// TIA Portal project "Ex2-PickAndPlace" (V16)
// The pick and place project

(* hardware
DEVICE "S7-1200 station_1"  S7-1200 Station
   slot 0: "Rack_0"  S7-1200 Rack  Rack  V1.0
   slot 1: "PLC_1"  CPU 1215C DC/DC/Rly  6ES7 215-1HG40-0XB0  V4.4
*)

// ===== PLC "PLC_1"  CPU 1215C DC/DC/Rly =====

VAR_GLOBAL   // PLC tag table "Default tag table"
   "System_Byte" AT %MB254 : Byte;
   "FirstScan" AT %M254.0 : Bool;
   "DiagStatusUpdate" AT %M254.1 : Bool;
   "AlwaysTRUE" AT %M254.2 : Bool;
   "AlwaysFALSE" AT %M254.3 : Bool;
   "Clock_Byte" AT %MB255 : Byte;
   "Clock_10Hz" AT %M255.0 : Bool;
   "Clock_5Hz" AT %M255.1 : Bool;
   "Clock_2.5Hz" AT %M255.2 : Bool;
   "Clock_2Hz" AT %M255.3 : Bool;
   "Clock_1.25Hz" AT %M255.4 : Bool;
   "Clock_1Hz" AT %M255.5 : Bool;
   "Clock_0.625Hz" AT %M255.6 : Bool;
   "Clock_0.5Hz" AT %M255.7 : Bool;
END_VAR

// folder: DB's

DATA_BLOCK "FB_CM_DI_Sensor_DB"   // DB1
{ S7_Optimized_Access := 'FALSE' }
AUTHOR : GeertVG
FAMILY : S88
VERSION : 0.1
// stored: InstanceOfName FB_CM_DI_Sensor
"FB_CM_DI_Sensor"
BEGIN
END_DATA_BLOCK

DATA_BLOCK "FB_PE_StartStop_DB"   // DB11
{ S7_Optimized_Access := 'FALSE' }
AUTHOR : GeertVG
FAMILY : S88
VERSION : 0.1
// stored: InstanceOfName FB_PE_StartStop
"FB_PE_StartStop"
BEGIN
END_DATA_BLOCK

DATA_BLOCK "FB_PE_Reset_DB"   // DB12
{ S7_Optimized_Access := 'FALSE' }
AUTHOR : GeertVG
FAMILY : S88
VERSION : 0.1
// stored: InstanceOfName FB_PE_Reset
"FB_PE_Reset"
BEGIN
END_DATA_BLOCK

DATA_BLOCK "FB_CM_Lamp_DB"   // DB13
{ S7_Optimized_Access := 'FALSE' }
AUTHOR : GeertVG
FAMILY : S88
VERSION : 0.1
// stored: InstanceOfName FB_CM_Lamp
"FB_CM_Lamp"
BEGIN
END_DATA_BLOCK

// folder: (top level)

FUNCTION_BLOCK "S88"   // FB1, FBD
TITLE = S88
{ S7_Optimized_Access := 'TRUE' }
VERSION : 0.1
// S88 software model for the pick and place project
BEGIN

REGION Network 1: Control module sensor
END_REGION
END_FUNCTION_BLOCK

FUNCTION "FC_EM_PnP" : Void   // FC1, FBD
TITLE = Equipment module for the pick and place
{ S7_Optimized_Access := 'TRUE' }
VERSION : 0.1
// Equipment module following the S88 software model for the pick and place project
BEGIN

REGION Network 1: Control module sensor B1
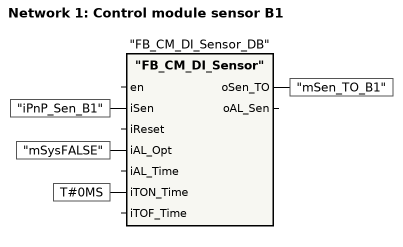
   "FB_CM_DI_Sensor_DB"(iSen := "iPnP_Sen_B1",   // "FB_CM_DI_Sensor"
                        iAL_Opt := "mSysFALSE",
                        iTON_Time := T#0MS,
                        oSen_TO => "mSen_TO_B1");
END_REGION
END_FUNCTION

FUNCTION "FC_EM_CC1" : Void   // FC2, FBD
TITLE = Circuit board 1
{ S7_Optimized_Access := 'TRUE' }
VERSION : 0.1
// This cicruit board handles the start and stop instruction. Lamps are being controlled here as well
BEGIN

REGION Network 1: Procedure element start stop
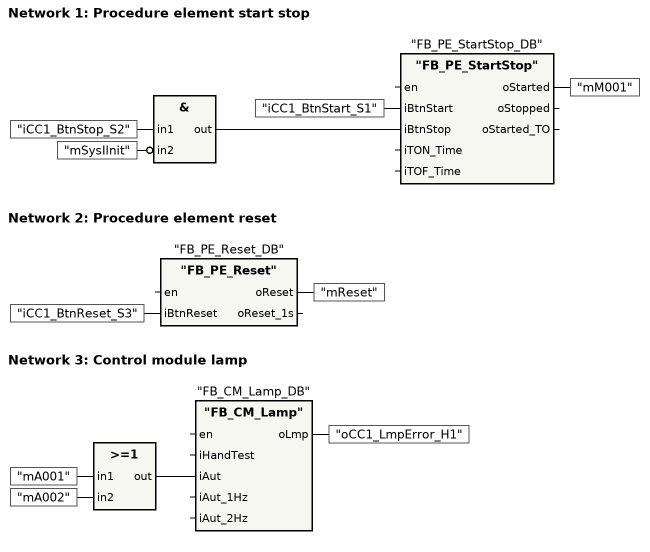
   "FB_PE_StartStop_DB"(iBtnStart := "iCC1_BtnStart_S1",   // "FB_PE_StartStop"
                        iBtnStop := "iCC1_BtnStop_S2" AND NOT "mSysIlnit",
                        oStarted => "mM001");
END_REGION

REGION Network 2: Procedure element reset
   "FB_PE_Reset_DB"(iBtnReset := "iCC1_BtnReset_S3", oReset => "mReset");   // "FB_PE_Reset"
END_REGION

REGION Network 3: Control module lamp
   "FB_CM_Lamp_DB"(iAut := "mA001" OR "mA002", oLmp => "oCC1_LmpError_H1");   // "FB_CM_Lamp"
END_REGION
END_FUNCTION

ORGANIZATION_BLOCK "Main"   // OB1, FBD, ProgramCycle
TITLE = "Main Program Sweep (Cycle)"
{ S7_Optimized_Access := 'TRUE' }
VERSION : 0.1
   VAR_INPUT
      Initial_Call : Bool;   // Initial call of this OB
      Remanence : Bool;   // =True, if remanent data are available
   END_VAR
BEGIN

REGION Network 1
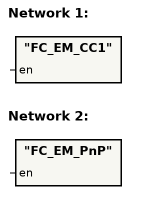
   "FC_EM_CC1"();
END_REGION

REGION Network 2
   "FC_EM_PnP"();
END_REGION
END_ORGANIZATION_BLOCK

// folder: Control modules (CM)

FUNCTION_BLOCK "FB_CM_DI_Sensor"   // FB10, FBD
TITLE = Control module digital sensor
{ S7_Optimized_Access := 'FALSE' }
AUTHOR : GeertVG
FAMILY : S88
VERSION : 0.1
// A control modul digital sensor processes the signal coming from a digital sensor and can delay a signal with the use of a rise- or a switch-off delay and/or in case a sensor gets activated to activate an alarm.
   VAR_INPUT
      iSen : Bool;   // Sensor
      iReset : Bool;   // Reset alarm
      iAL_Opt : Bool;   // Alarm option enabled if TRUE
      iAL_Time : Time;   // Rise-delay sensor alarm
      iTON_Time : Time;   // Sensor rise-delay
      iTOF_Time : Time;   // Sensor switch-off delay
   END_VAR
   VAR_OUTPUT
      oSen_TO : Bool;   // Sensor after delay
      oAL_Sen : Bool;   // Alarm sensor activated
   END_VAR
   VAR
      sTON_AL : TON_TIME;   // Rise-delay for oAL_sen
      sTON : TON_TIME;   // Rise-delay for oSen_TO
      sTOF : TOF_TIME;   // Switch-off delay for oSen_TO
      sAL_Sen : Bool;   // Sensor alarm
      sTON_Aon : Bool;
   END_VAR
BEGIN

REGION Network 1: Rise-delay for the activated alarm sensor
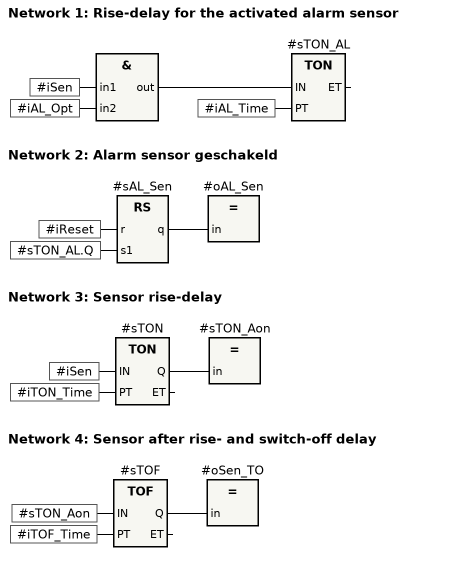
   #sTON_AL(IN := #iSen AND #iAL_Opt, PT := #iAL_Time);   // TON
END_REGION

REGION Network 2: Alarm sensor geschakeld
   IF #iReset THEN
       #sAL_Sen := FALSE;   // RS flip-flop
   END_IF;
   IF #sTON_AL.Q THEN #sAL_Sen := TRUE; END_IF;
   #oAL_Sen := #sAL_Sen;
END_REGION

REGION Network 3: Sensor rise-delay
   #sTON(IN := #iSen, PT := #iTON_Time);   // TON
   #sTON_Aon := #sTON.Q;
END_REGION

REGION Network 4: Sensor after rise- and switch-off delay
   #sTOF(IN := #sTON_Aon, PT := #iTOF_Time);   // TOF
   #oSen_TO := #sTOF.Q;
END_REGION
END_FUNCTION_BLOCK

FUNCTION_BLOCK "FB_CM_Lamp"   // FB16, FBD
TITLE = Control module lamp
{ S7_Optimized_Access := 'FALSE' }
AUTHOR : GeertVG
FAMILY : S88
VERSION : 0.1
// A control module lamp will actiavte a lamp (if chosen blinking). Also the possibility of testing the lamp with the use of the test input.
   VAR_INPUT
      iHandTest : Bool;   // Lamptest
      iAut : Bool;   // Lamp continue activation
      iAut_1Hz : Bool;   // Lamp blinking slowly
      iAut_2Hz : Bool;   // Lamp blinking fast
   END_VAR
   VAR_OUTPUT
      oLmp : Bool;   // Lamp
   END_VAR
   VAR
      sTON_1Hz_On : TON_TIME;   // 1 Hz timer lamp on
      sTON_1Hz_Off : TON_TIME;   // 1 Hz timer lamp off
      sTON_2Hz_On : TON_TIME;   // 2 Hz timer lamp on
      sTON_2Hz_Off : TON_TIME;   // 2 Hz timer lamp off
      sOn_1Hz : Bool;
      sOff_1Hz : Bool;
      sOn_2Hz : Bool;
      sOff_2Hz : Bool;
   END_VAR
BEGIN

REGION Network 1: Blinkcicuit 1Hz
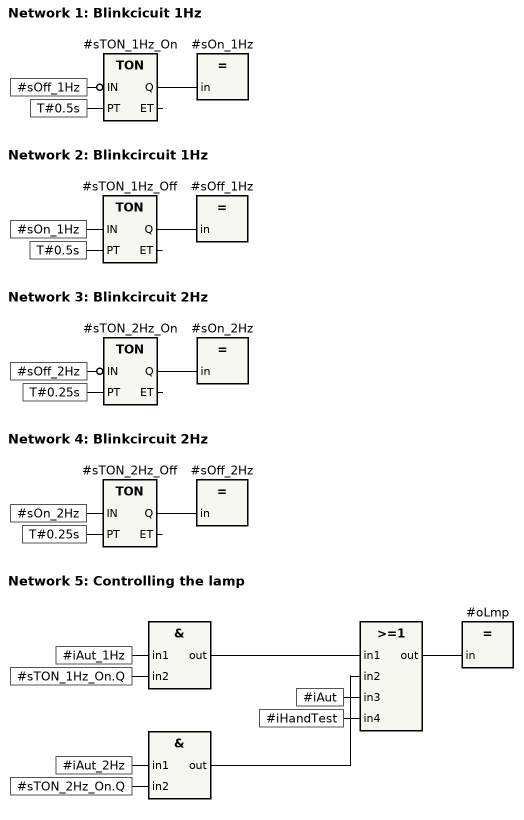
   #sTON_1Hz_On(IN := NOT #sOff_1Hz, PT := T#0.5s);   // TON
   #sOn_1Hz := #sTON_1Hz_On.Q;
END_REGION

REGION Network 2: Blinkcircuit 1Hz
   #sTON_1Hz_Off(IN := #sOn_1Hz, PT := T#0.5s);   // TON
   #sOff_1Hz := #sTON_1Hz_Off.Q;
END_REGION

REGION Network 3: Blinkcircuit 2Hz
   #sTON_2Hz_On(IN := NOT #sOff_2Hz, PT := T#0.25s);   // TON
   #sOn_2Hz := #sTON_2Hz_On.Q;
END_REGION

REGION Network 4: Blinkcircuit 2Hz
   #sTON_2Hz_Off(IN := #sOn_2Hz, PT := T#0.25s);   // TON
   #sOff_2Hz := #sTON_2Hz_Off.Q;
END_REGION

REGION Network 5: Controlling the lamp
   #oLmp := (#iAut_1Hz AND #sTON_1Hz_On.Q) OR (#iAut_2Hz AND #sTON_2Hz_On.Q) OR #iAut OR #iHandTest;
END_REGION
END_FUNCTION_BLOCK

// folder: Procedure Elements (PE)

FUNCTION_BLOCK "FB_PE_StartStop"   // FB30, FBD
TITLE = Start-Stop procedure element
{ S7_Optimized_Access := 'FALSE' }
AUTHOR : GeertVG
FAMILY : S88
VERSION : 0.1
// A start-stop is used to start and stop actuators and/or the automatic process of a installation/machine (or parts of it).
   VAR_INPUT
      iBtnStart : Bool;   // Start button(NO)
      iBtnStop : Bool;   // Stop button (NC)
      iTON_Time : Time;   // Opkomvertraging voor oGestart_TO
      iTOF_Time : Time;   // Afvalvertraging voor oGestart_TO
   END_VAR
   VAR_OUTPUT
      oStarted : Bool;   // Started
      oStopped : Bool;   // Stopped
      oStarted_TO : Bool;   // Started with a rise or off-delay
   END_VAR
   VAR
      sStarted : Bool;   // Started
      sPfBtnStart : Bool;   // Rising flank of iBtnStart
      sTON_Started : Bool;   // Start with on-delay
      sTON : TON_TIME;   // On-delay
      sTOF : TOF_TIME;   // Off-delay
   END_VAR
   VAR_TEMP   // added for the SCL form of the ladder/FBD networks
      _w1 : Bool;
   END_VAR
BEGIN

REGION Network 1: Start-stop using a FlipFlop instruction
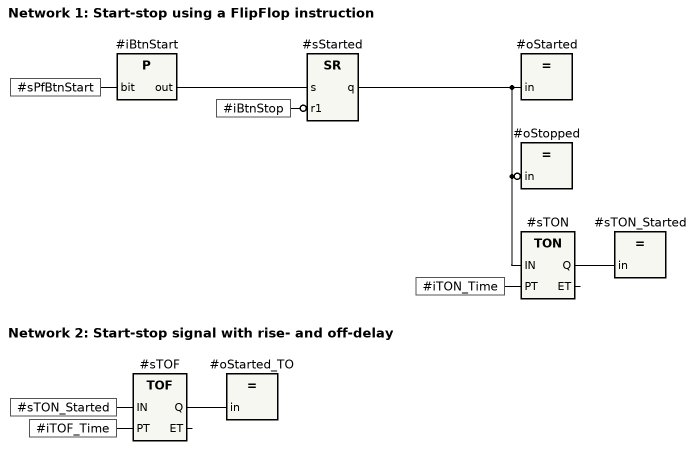
   #_w1 := #iBtnStart AND NOT #sPfBtnStart;   // rising edge of #iBtnStart
   #sPfBtnStart := #iBtnStart;
   IF #_w1 THEN
       #sStarted := TRUE;   // SR flip-flop
   END_IF;
   IF NOT #iBtnStop THEN #sStarted := FALSE; END_IF;
   #oStarted := #sStarted;
   #oStopped := NOT #sStarted;
   #sTON(IN := #sStarted, PT := #iTON_Time);   // TON
   #sTON_Started := #sTON.Q;
END_REGION

REGION Network 2: Start-stop signal with rise- and off-delay
   #sTOF(IN := #sTON_Started, PT := #iTOF_Time);   // TOF
   #oStarted_TO := #sTOF.Q;
END_REGION
END_FUNCTION_BLOCK

FUNCTION_BLOCK "FB_PE_Reset"   // FB31, FBD
TITLE = Reset procedure element
{ S7_Optimized_Access := 'FALSE' }
AUTHOR : GeertVG
FAMILY : S88
VERSION : 0.1
// The reset procedure is commonly used to create a controlled reset signal. Controlled because the signal is coming from a for example. an electyrical reset button (NO contact) can contain errors like a shortcircuit, the bridging of a signal and a bad/ fake contact.
   VAR_INPUT
      iBtnReset : Bool;   // Reset button
   END_VAR
   VAR_OUTPUT
      oReset : Bool;   // Checked reset signal (1 cyclus)
      oReset_1s : Bool;   // Checked reset signal (1s)
   END_VAR
   VAR
      sNfReset : Bool;
      sTON_Max : TON_TIME;   // Max. time that the button can be pressed
      sTON_Min : TON_TIME;   // Min. time that the button can be pressed
      sTP : TP_TIME;   // Checked reset time off 1s
   END_VAR
   VAR_TEMP   // added for the SCL form of the ladder/FBD networks
      _w1 : Bool;
   END_VAR
BEGIN

REGION Network 1: Max. time
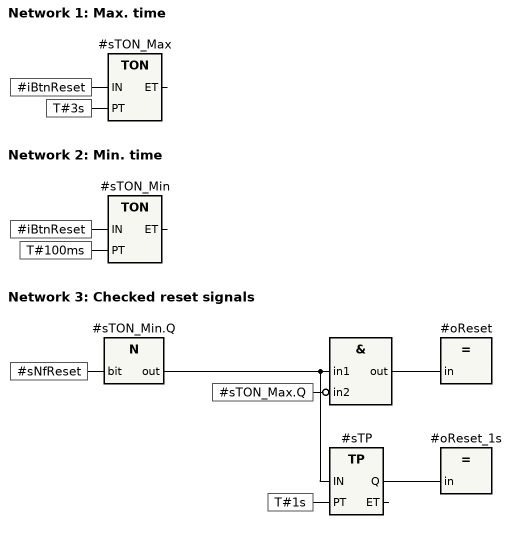
   #sTON_Max(IN := #iBtnReset, PT := T#3s);   // TON
END_REGION

REGION Network 2: Min. time
   #sTON_Min(IN := #iBtnReset, PT := T#100ms);   // TON
END_REGION

REGION Network 3: Checked reset signals
   #_w1 := NOT #sTON_Min.Q AND #sNfReset;   // falling edge of #sTON_Min.Q
   #sNfReset := #sTON_Min.Q;
   #oReset := #_w1 AND NOT #sTON_Max.Q;
   #sTP(IN := #_w1, PT := T#1s);   // TP
   #oReset_1s := #sTP.Q;
END_REGION
END_FUNCTION_BLOCK

// ===== library types =====

// folder: Control modules (CM)

FUNCTION_BLOCK "FB_CM_AI_Sensor"   // FB11, FBD
TITLE = Control module analogesensor
{ S7_Optimized_Access := 'FALSE' }
AUTHOR : GeertVG
FAMILY : S88
VERSION : 0.1
// The control module analog sensor converts a measured number to a SI-Unit
// In case of incorrect operation of the sensor a alarm will be created.
   VAR_INPUT
      iSen : Int;   // Measured value
      iReset : Bool;   // Reset alarm
      iHiLim : Real;   // The upper measurelimit of the sensor
      iLoLim : Real;   // The lower measurelimit of the sensor
      iUniOpt : Bool;   // 1 = Unipolair / 0 = Bipolair
   END_VAR
   VAR_OUTPUT
      oX : Real;   // The measured value gets converted to a SI-Unit
      oAL_Sen : Bool;   // Alarm sensor defect
   END_VAR
   VAR
      sAL_Sen : Bool;   // Alarm sensor defect
      sSen_DINT : DInt;   // Measured Value
      sMIN : DInt;   // Under Limit
      sNORM_Counter : DInt;
      sNORM_Denominator : DInt;
      sNORM_Counter_REAL : Real;
      sNORM_Denominator_REAL : Real;
      sNORM_X : Real;
      sSCALE_MeasureRange : Real;
      sSCALE_X : Real;
   END_VAR
BEGIN

REGION Network 1: Conversion sensor
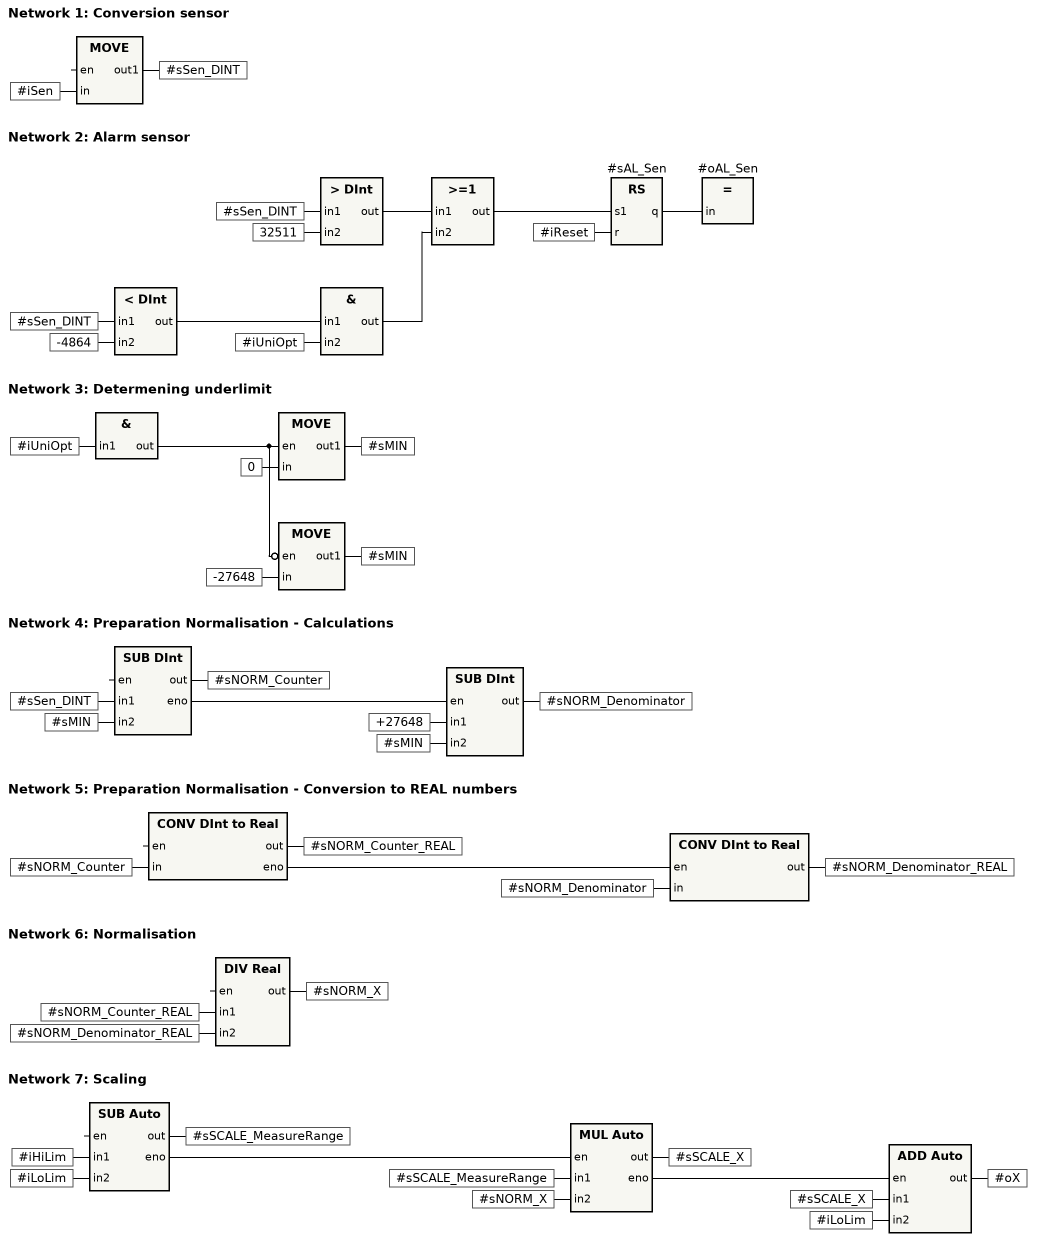
   #sSen_DINT := #iSen;
END_REGION

REGION Network 2: Alarm sensor
   IF #iReset THEN
       #sAL_Sen := FALSE;   // RS flip-flop
   END_IF;
   IF (#sSen_DINT > 32511) OR ((#sSen_DINT < (-4864)) AND #iUniOpt) THEN #sAL_Sen := TRUE; END_IF;
   #oAL_Sen := #sAL_Sen;
END_REGION

REGION Network 3: Determening underlimit
   IF #iUniOpt THEN #sMIN := 0; END_IF;
   IF NOT #iUniOpt THEN #sMIN := -27648; END_IF;
END_REGION

REGION Network 4: Preparation Normalisation - Calculations
   #sNORM_Counter := #sSen_DINT - #sMIN;
   #sNORM_Denominator := +27648 - #sMIN;
END_REGION

REGION Network 5: Preparation Normalisation - Conversion to REAL numbers
   #sNORM_Counter_REAL := DINT_TO_REAL(#sNORM_Counter);
   #sNORM_Denominator_REAL := DINT_TO_REAL(#sNORM_Denominator);
END_REGION

REGION Network 6: Normalisation
   #sNORM_X := #sNORM_Counter_REAL / #sNORM_Denominator_REAL;
END_REGION

REGION Network 7: Scaling
   #sSCALE_MeasureRange := #iHiLim - #iLoLim;
   #sSCALE_X := #sSCALE_MeasureRange * #sNORM_X;
   #oX := #sSCALE_X + #iLoLim;
END_REGION
END_FUNCTION_BLOCK

FUNCTION_BLOCK "FB_CM_DOL"   // FB12, FBD
TITLE = Control module asynchronous motor 1 direction 1 speed
{ S7_Optimized_Access := 'FALSE' }
AUTHOR : GeertVG
FAMILY : S88
VERSION : 0.1
// A control module asynchronous motor 1 direction 1 speed controls the management of a 3-phase asynchronous motor with a motor circuit breaker and one contactor. The control module is provided with a hand workmode, an automatic workingmode, moter circuit breaker alarm and an enable.
   VAR_INPUT
      iEnable : Bool;
      iReset : Bool;
      iMcb : Bool;
      iModeHand : Bool;
      iHandOn : Bool;
      iHandOff : Bool;
      iAut : Bool;
      iTON_Time : Time;
      iTOF_Time : Time;
   END_VAR
   VAR_OUTPUT
      oCon : Bool;
      oAL_Mcb : Bool;
   END_VAR
   VAR
      sAl_Mcb : Bool;
      sStarted : Bool;
      sTON_Started : Bool;
      sTO_Started : Bool;
      sTOF : TOF_TIME;
      sTON : TON_TIME;
   END_VAR
BEGIN

REGION Network 1: Alarm motor circuit breaker
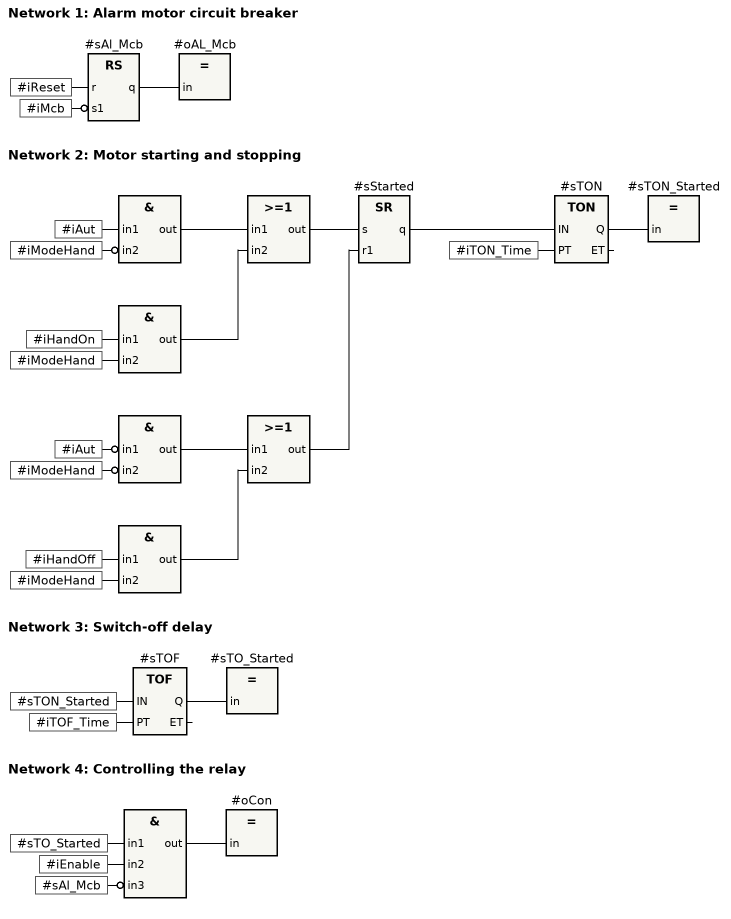
   IF #iReset THEN
       #sAl_Mcb := FALSE;   // RS flip-flop
   END_IF;
   IF NOT #iMcb THEN #sAl_Mcb := TRUE; END_IF;
   #oAL_Mcb := #sAl_Mcb;
END_REGION

REGION Network 2: Motor starting and stopping
   IF (#iAut AND NOT #iModeHand) OR (#iHandOn AND #iModeHand) THEN
       #sStarted := TRUE;   // SR flip-flop
   END_IF;
   IF (NOT #iAut AND NOT #iModeHand) OR (#iHandOff AND #iModeHand) THEN #sStarted := FALSE; END_IF;
   #sTON(IN := #sStarted, PT := #iTON_Time);   // TON
   #sTON_Started := #sTON.Q;
END_REGION

REGION Network 3: Switch-off delay
   #sTOF(IN := #sTON_Started, PT := #iTOF_Time);   // TOF
   #sTO_Started := #sTOF.Q;
END_REGION

REGION Network 4: Controlling the relay
   #oCon := #sTO_Started AND #iEnable AND NOT #sAl_Mcb;
END_REGION
END_FUNCTION_BLOCK

FUNCTION_BLOCK "FB_CM_DOLRev"   // FB13, FBD
TITLE = Control module asynchronous motor 2 directions 1 speed
{ S7_Optimized_Access := 'FALSE' }
AUTHOR : GeertVG
FAMILY : S88
VERSION : 0.1
// A control module asynchronous motor 2 directions 1 speed controls the management of a 3-phase asynchronous motor with a motor circuit breaker and 2 relays to turn around the turn direction. The control module is provided with a hand workmode, an automatic workingmode, moter circuit breaker alarm and an enable.
   VAR_INPUT
      iEnable : Bool;
      iReset : Bool;
      iMcb : Bool;
      iModeHand : Bool;
      iHandR : Bool;
      iHandL : Bool;
      iHandOff : Bool;
      iAutR : Bool;
      iAutL : Bool;
      iTOF_Time : Time;
   END_VAR
   VAR_OUTPUT
      oConR : Bool;
      oConL : Bool;
      oAL_Mcb : Bool;
   END_VAR
   VAR
      sAl_Mcb : Bool;
      sStartedR : Bool;
      sStartedL : Bool;
      sTOF_R : TOF_TIME;
      sTOF_L : TOF_TIME;
   END_VAR
   VAR_TEMP   // added for the SCL form of the ladder/FBD networks
      _w1 : Bool;
   END_VAR
BEGIN

REGION Network 1: Alarm motor circuit breaker
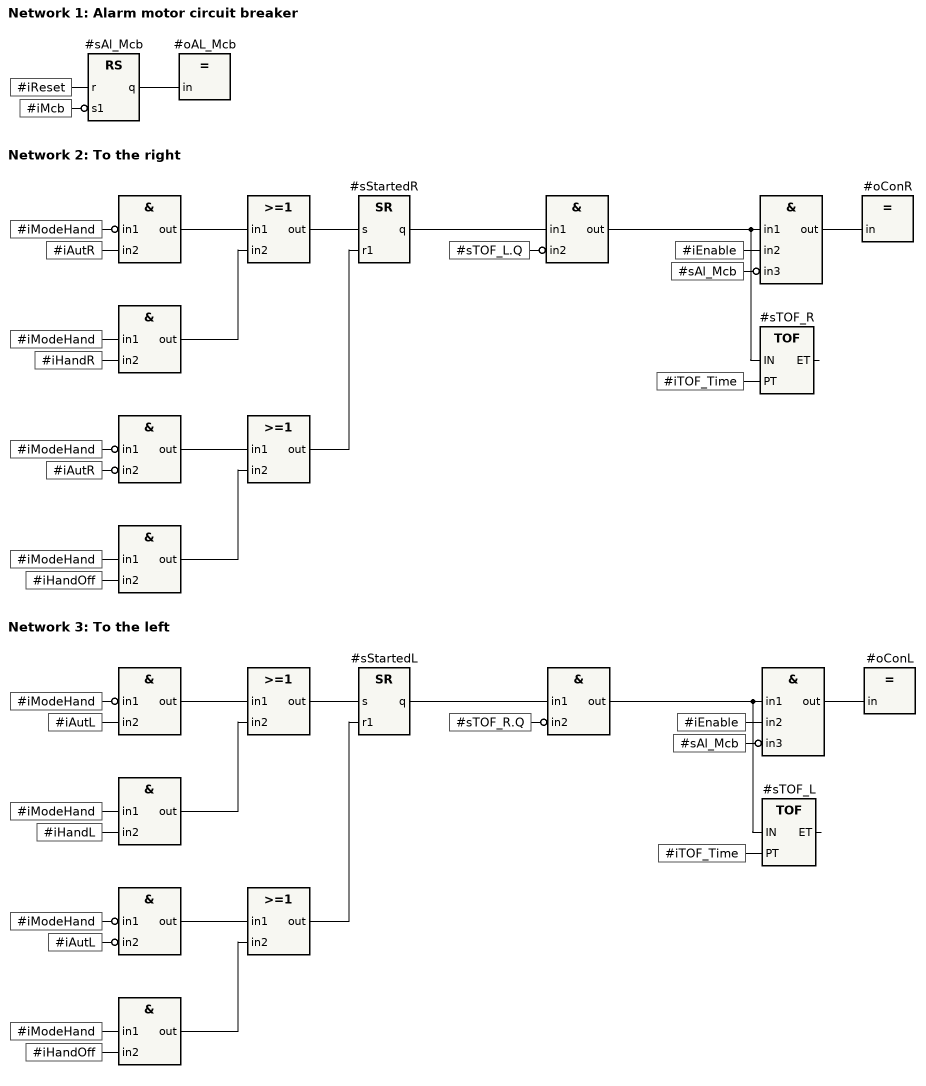
   IF #iReset THEN
       #sAl_Mcb := FALSE;   // RS flip-flop
   END_IF;
   IF NOT #iMcb THEN #sAl_Mcb := TRUE; END_IF;
   #oAL_Mcb := #sAl_Mcb;
END_REGION

REGION Network 2: To the right
   IF (NOT #iModeHand AND #iAutR) OR (#iModeHand AND #iHandR) THEN
       #sStartedR := TRUE;   // SR flip-flop
   END_IF;
   IF (NOT #iModeHand AND NOT #iAutR) OR (#iModeHand AND #iHandOff) THEN #sStartedR := FALSE; END_IF;
   #_w1 := #sStartedR AND NOT #sTOF_L.Q;
   #oConR := #_w1 AND #iEnable AND NOT #sAl_Mcb;
   #sTOF_R(IN := #_w1, PT := #iTOF_Time);   // TOF
END_REGION

REGION Network 3: To the left
   IF (NOT #iModeHand AND #iAutL) OR (#iModeHand AND #iHandL) THEN
       #sStartedL := TRUE;   // SR flip-flop
   END_IF;
   IF (NOT #iModeHand AND NOT #iAutL) OR (#iModeHand AND #iHandOff) THEN #sStartedL := FALSE; END_IF;
   #_w1 := #sStartedL AND NOT #sTOF_R.Q;
   #oConL := #_w1 AND #iEnable AND NOT #sAl_Mcb;
   #sTOF_L(IN := #_w1, PT := #iTOF_Time);   // TOF
END_REGION
END_FUNCTION_BLOCK

FUNCTION_BLOCK "FB_CM_Valve"   // FB14, FBD
TITLE = Control module valve
{ S7_Optimized_Access := 'FALSE' }
AUTHOR : GeertVG
FAMILY : S88
VERSION : 0.1
// A control module valve is used to control a electromechanical pressured air valve or electormechanical valve.
   VAR_INPUT
      iEnable : Bool;
      iModeHand : Bool;
      iHand_1 : Bool;
      iHand_0 : Bool;
      iAut_1 : Bool;
      iAut_0 : Bool;
   END_VAR
   VAR_OUTPUT
      oVal_1 : Bool;
      oVal_0 : Bool;
   END_VAR
   VAR
      sVal_1 : Bool;
      sVal_0 : Bool;
   END_VAR
BEGIN

REGION Network 1: Valve p(ositive) memory (TRUE condition)
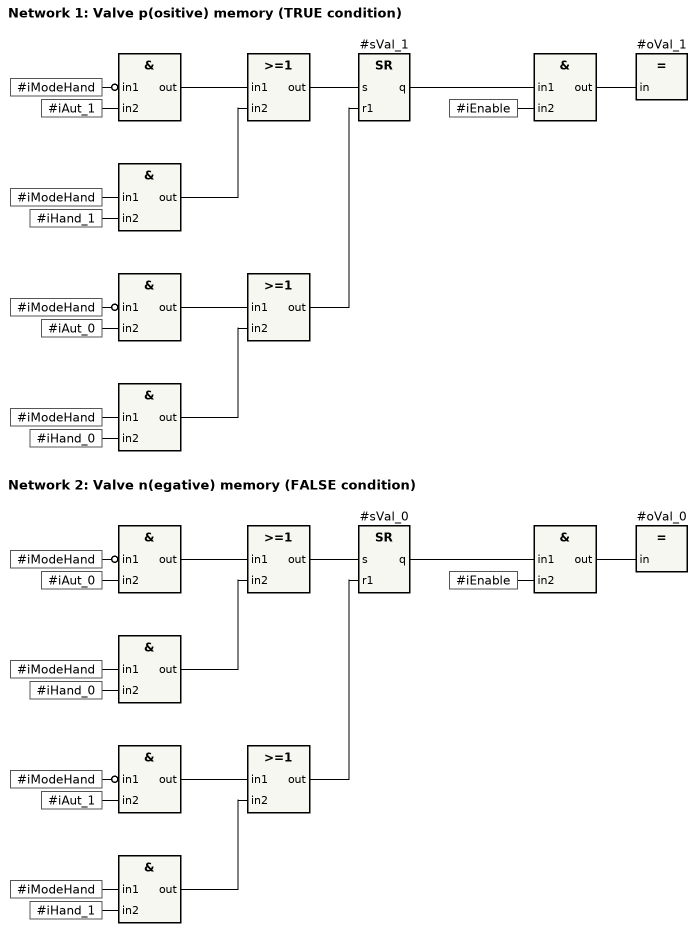
   IF (NOT #iModeHand AND #iAut_1) OR (#iModeHand AND #iHand_1) THEN
       #sVal_1 := TRUE;   // SR flip-flop
   END_IF;
   IF (NOT #iModeHand AND #iAut_0) OR (#iModeHand AND #iHand_0) THEN #sVal_1 := FALSE; END_IF;
   #oVal_1 := #sVal_1 AND #iEnable;
END_REGION

REGION Network 2: Valve n(egative) memory (FALSE condition)
   IF (NOT #iModeHand AND #iAut_0) OR (#iModeHand AND #iHand_0) THEN
       #sVal_0 := TRUE;   // SR flip-flop
   END_IF;
   IF (NOT #iModeHand AND #iAut_1) OR (#iModeHand AND #iHand_1) THEN #sVal_0 := FALSE; END_IF;
   #oVal_0 := #sVal_0 AND #iEnable;
END_REGION
END_FUNCTION_BLOCK

FUNCTION_BLOCK "FB_CM_Relay"   // FB15, FBD
TITLE = Control module relay
{ S7_Optimized_Access := 'FALSE' }
AUTHOR : GeertVG
FAMILY : S88
VERSION : 0.1
// A control module relay gets used to control a relay that isn't used in a motorcircuit.
   VAR_INPUT
      iEnable : Bool;
      iModeHand : Bool;
      iHandOn : Bool;
      iHandOff : Bool;
      iAut : Bool;
      iTON_Time : Time;
      iTOF_Time : Time;
   END_VAR
   VAR_OUTPUT
      oCon : Bool;
   END_VAR
   VAR
      sStarted : Bool;
      sTON_Started : Bool;
      STO_Started : Bool;
      sTON : TON_TIME;
      sTOF : TOF_TIME;
   END_VAR
BEGIN

REGION Network 1: Start stop circuit
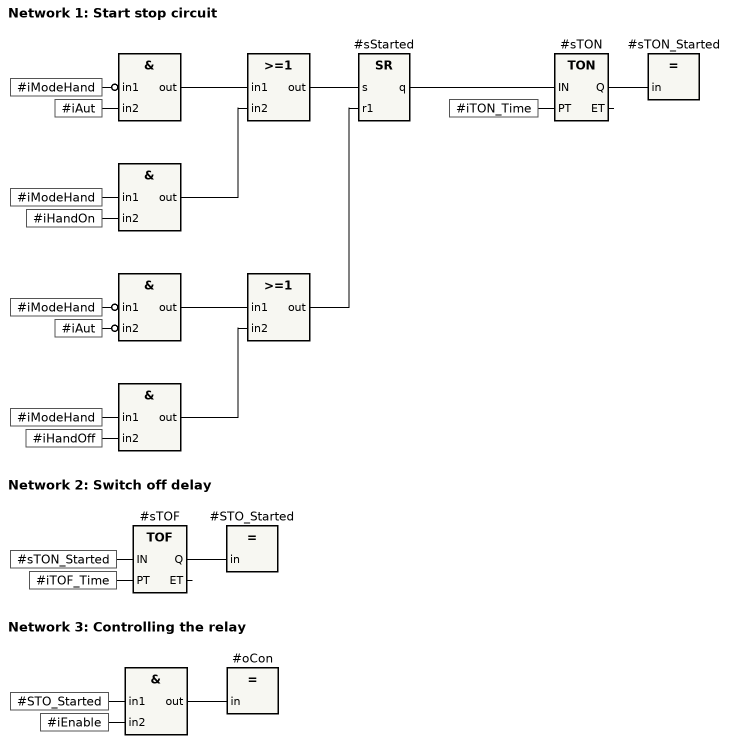
   IF (NOT #iModeHand AND #iAut) OR (#iModeHand AND #iHandOn) THEN
       #sStarted := TRUE;   // SR flip-flop
   END_IF;
   IF (NOT #iModeHand AND NOT #iAut) OR (#iModeHand AND #iHandOff) THEN #sStarted := FALSE; END_IF;
   #sTON(IN := #sStarted, PT := #iTON_Time);   // TON
   #sTON_Started := #sTON.Q;
END_REGION

REGION Network 2: Switch off delay
   #sTOF(IN := #sTON_Started, PT := #iTOF_Time);   // TOF
   #STO_Started := #sTOF.Q;
END_REGION

REGION Network 3: Controlling the relay
   #oCon := #STO_Started AND #iEnable;
END_REGION
END_FUNCTION_BLOCK

// folder: Procedure Elementen (PE)

FUNCTION_BLOCK "FB_PE_ON-OFF"   // FB32, FBD
TITLE = Procedure element on-off controller with hysteresis
{ S7_Optimized_Access := 'FALSE' }
AUTHOR : GeertVG
FAMILY : S88
VERSION : 0.1
// A on-off controller with hysteresis is commonly used in an on-off circuit to switch an actuator on or off in fuction of a measured nature unit (= the measured value X) and a desired nature unit ( = Lop manipulated value Y).
   VAR_INPUT
      iOn : Bool;   // Controller on- or off-switch
      iX : Real;   // Measured value
      iW : Real;   // Loop manipulated value
      iH : Real;   // Hysteresis
   END_VAR
   VAR_OUTPUT
      oY : Bool;   // Setpoint
      oY_NOT : Bool;   // Setpoint inverted
   END_VAR
   VAR
      sOn : Bool;
   END_VAR
   VAR_TEMP
      xHystDiv2 : Real;   // Hysteresis / 2.0
      xWAddHystDiv2 : Real;   // Loop manipulated value + Hysteresis / 2.0
      xWSubHystDiv2 : Real;   // Loop manipulated value - Hysteresis / 2.0
   END_VAR
BEGIN

REGION Network 1: Switchpoints
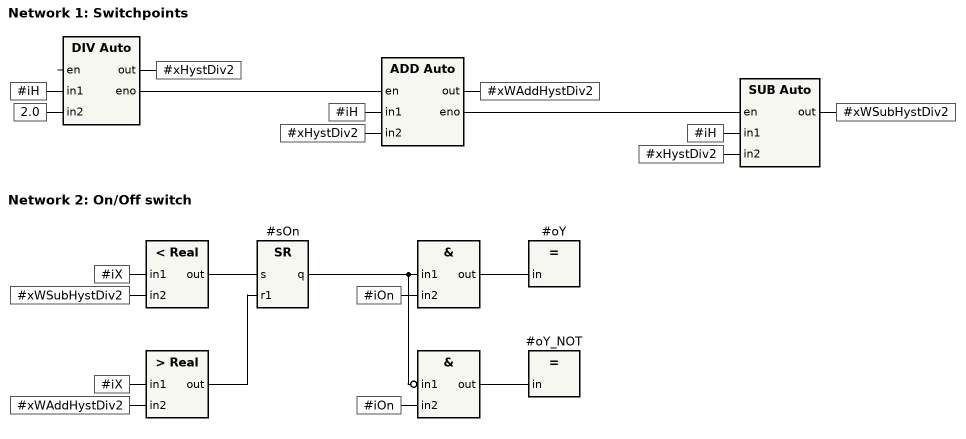
   #xHystDiv2 := #iH / 2.0;
   #xWAddHystDiv2 := #iH + #xHystDiv2;
   #xWSubHystDiv2 := #iH - #xHystDiv2;
END_REGION

REGION Network 2: On/Off switch
   IF #iX < #xWSubHystDiv2 THEN
       #sOn := TRUE;   // SR flip-flop
   END_IF;
   IF #iX > #xWAddHystDiv2 THEN #sOn := FALSE; END_IF;
   #oY := #sOn AND #iOn;
   #oY_NOT := NOT #sOn AND #iOn;
END_REGION
END_FUNCTION_BLOCK